// SIMATIC S7-200 project (STEP 7-Micro/WIN), CPU 226 REL 02.01

SYMBOL_TABLE 用户定义1
mAuto            I0.0     // 自动循环模式
mPosDirection    I0.1     // 正转方向
mRun             I1.1     // 启动
mStop            I1.3     // 停止
mStoped          I1.5     // 停止状态
rRunStop         Q0.0     // 启停输出K1
rDirection       Q0.2     // 方向输出K2
rBreak           Q0.5     // 制动输出K4
cmdRun           M0.2     // 运行指令
cmdDirPos        M0.3     // 方向指令1为正转
cmdModAuto       M0.4     // 手自动模式1为自动
TMP              M0.1
PosDuringAuto    M0.5     // 自动运行时切换方向触发
TMP1             M0.6
TMP2             M0.7
mAin             AIW0     // 用于设定时间的模拟量输入
END_SYMBOL_TABLE

SYMBOL_TABLE S7-200 符号
Always_On        SM0.0    // 始终接通为 ON
First_Scan_On    SM0.1    // 仅第一个扫描周期中接通为 ON
END_SYMBOL_TABLE

ORGANIZATION_BLOCK 主程序:OB1
TITLE=
VAR
AllTime:INT;	// LW0 
PosTime:INT;	// LW2 
END_VAR
BEGIN
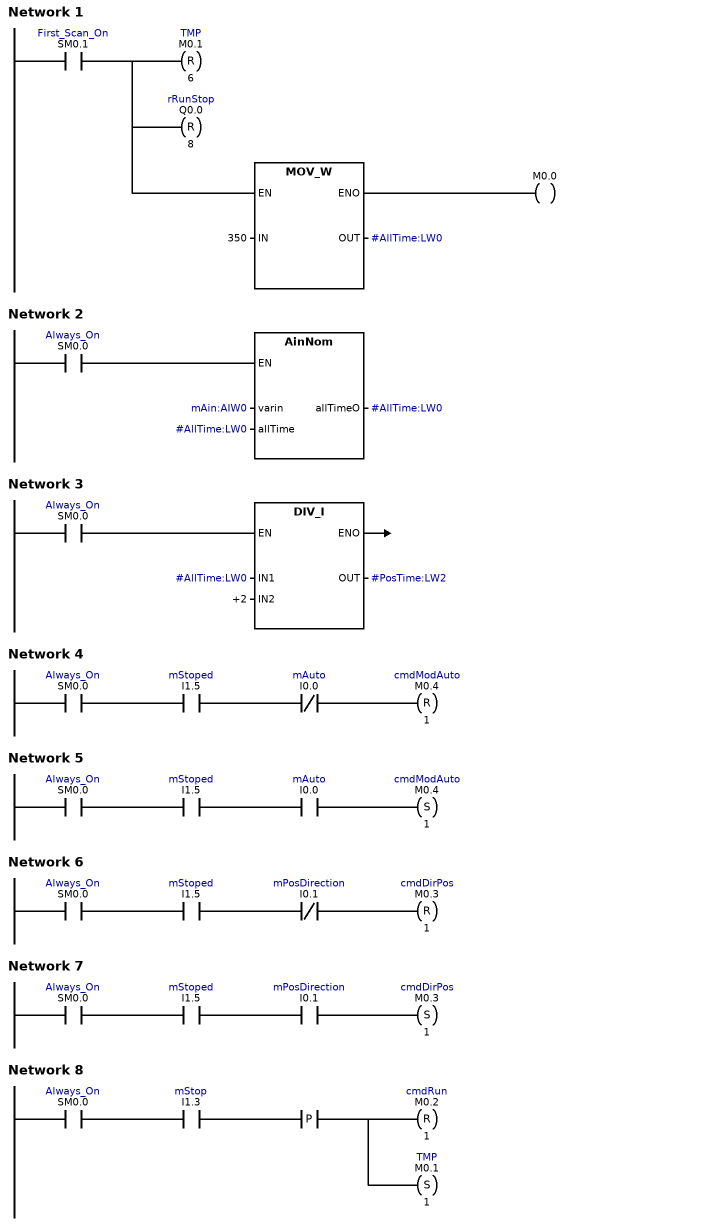
Network 1
LD     First_Scan_On:SM0.1
R      TMP:M0.1, 6
R      rRunStop:Q0.0, 8
MOVW   350, #AllTime:LW0
AENO
=      M0.0
Network 2
LD     Always_On:SM0.0
CALL   AinNom:SBR1, mAin:AIW0, #AllTime:LW0, #AllTime:LW0
Network 3
LD     Always_On:SM0.0
MOVW   #AllTime:LW0, #PosTime:LW2
/I     +2, #PosTime:LW2
Network 4
LD     Always_On:SM0.0
A      mStoped:I1.5
AN     mAuto:I0.0
R      cmdModAuto:M0.4, 1
Network 5
LD     Always_On:SM0.0
A      mStoped:I1.5
A      mAuto:I0.0
S      cmdModAuto:M0.4, 1
Network 6
LD     Always_On:SM0.0
A      mStoped:I1.5
AN     mPosDirection:I0.1
R      cmdDirPos:M0.3, 1
Network 7
LD     Always_On:SM0.0
A      mStoped:I1.5
A      mPosDirection:I0.1
S      cmdDirPos:M0.3, 1
Network 8
LD     Always_On:SM0.0
A      mStop:I1.3
EU
R      cmdRun:M0.2, 1
S      TMP:M0.1, 1
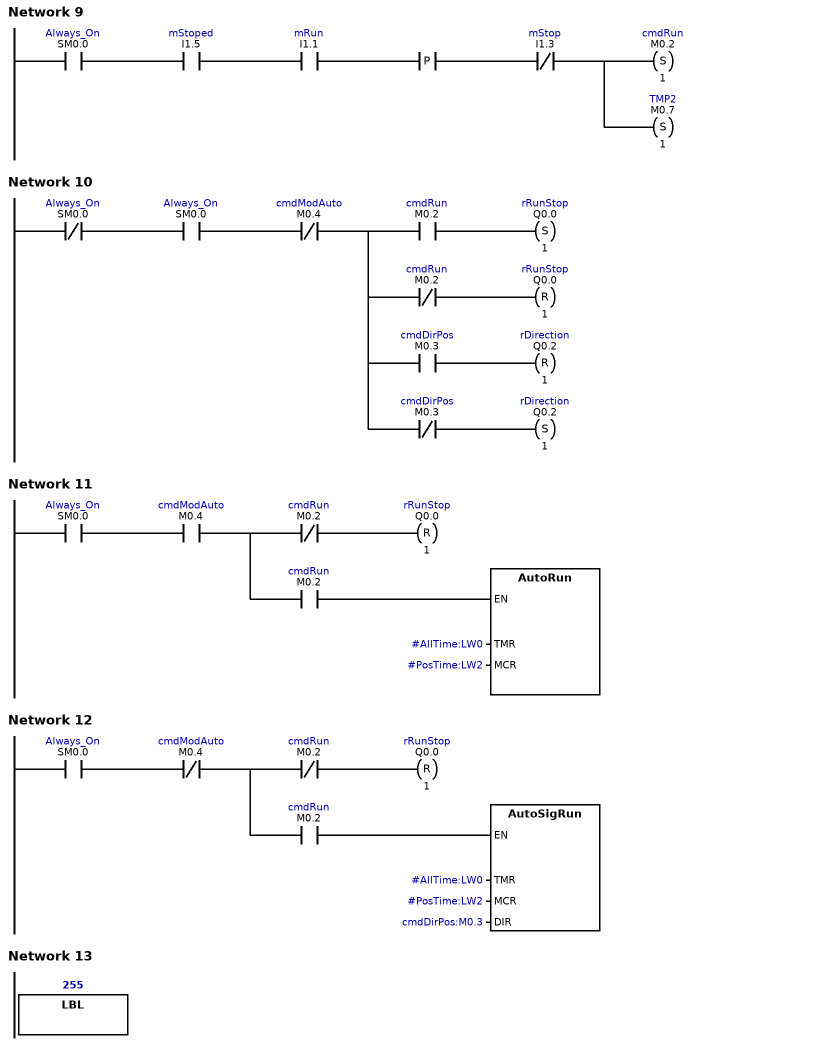
Network 9
LD     Always_On:SM0.0
A      mStoped:I1.5
A      mRun:I1.1
EU
AN     mStop:I1.3
S      cmdRun:M0.2, 1
S      TMP2:M0.7, 1
Network 10
LDN    Always_On:SM0.0
A      Always_On:SM0.0
AN     cmdModAuto:M0.4
LPS
A      cmdRun:M0.2
S      rRunStop:Q0.0, 1
LRD
AN     cmdRun:M0.2
R      rRunStop:Q0.0, 1
LRD
A      cmdDirPos:M0.3
R      rDirection:Q0.2, 1
LPP
AN     cmdDirPos:M0.3
S      rDirection:Q0.2, 1
Network 11
LD     Always_On:SM0.0
A      cmdModAuto:M0.4
LPS
AN     cmdRun:M0.2
R      rRunStop:Q0.0, 1
LPP
A      cmdRun:M0.2
CALL   AutoRun:SBR0, #AllTime:LW0, #PosTime:LW2
Network 12
LD     Always_On:SM0.0
AN     cmdModAuto:M0.4
LPS
AN     cmdRun:M0.2
R      rRunStop:Q0.0, 1
LPP
A      cmdRun:M0.2
CALL   AutoSigRun:SBR2, #AllTime:LW0, #PosTime:LW2, cmdDirPos:M0.3
Network 13
LBL    255
END_ORGANIZATION_BLOCK

SUBROUTINE_BLOCK AutoRun:SBR0
TITLE=子程序注释
VAR_INPUT
TMR:INT;	// LW0 
MCR:INT;	// LW2 
END_VAR
VAR
DET:INT;	// LW4 
END_VAR
BEGIN
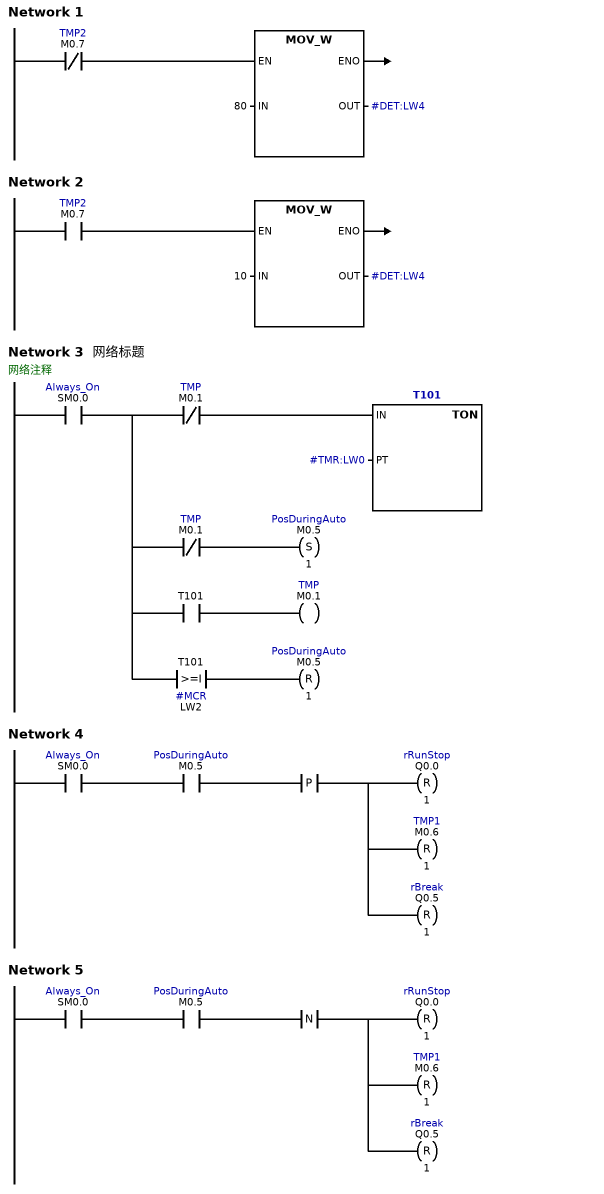
Network 1
LDN    TMP2:M0.7
MOVW   80, #DET:LW4
Network 2
LD     TMP2:M0.7
MOVW   10, #DET:LW4
Network 3 // 网络标题
// 网络注释
LD     Always_On:SM0.0
LPS
AN     TMP:M0.1
TON    T101, #TMR:LW0
LRD
AN     TMP:M0.1
S      PosDuringAuto:M0.5, 1
LRD
A      T101
=      TMP:M0.1
LPP
AW>=   T101, #MCR:LW2
R      PosDuringAuto:M0.5, 1
Network 4
LD     Always_On:SM0.0
A      PosDuringAuto:M0.5
EU
R      rRunStop:Q0.0, 1
R      TMP1:M0.6, 1
R      rBreak:Q0.5, 1
Network 5
LD     Always_On:SM0.0
A      PosDuringAuto:M0.5
ED
R      rRunStop:Q0.0, 1
R      TMP1:M0.6, 1
R      rBreak:Q0.5, 1
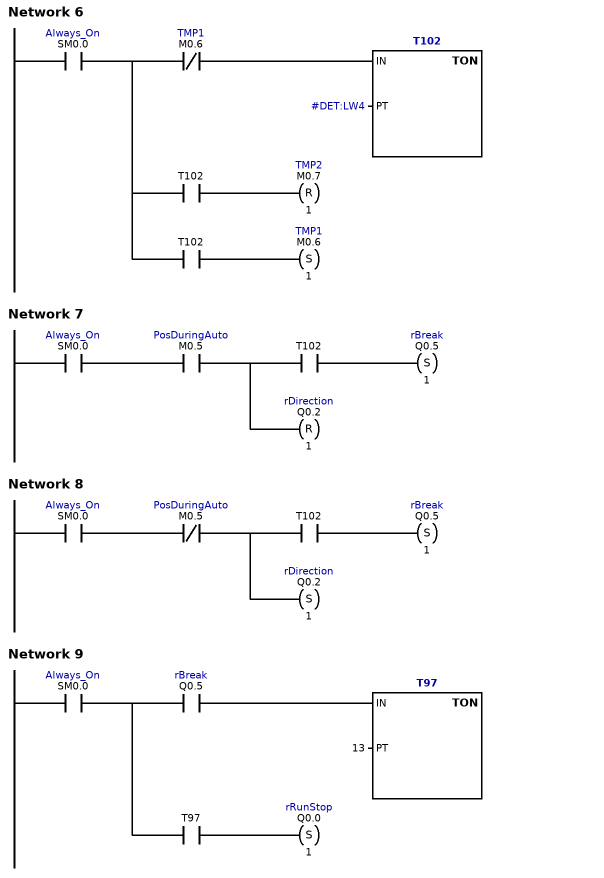
Network 6
LD     Always_On:SM0.0
LPS
AN     TMP1:M0.6
TON    T102, #DET:LW4
LRD
A      T102
R      TMP2:M0.7, 1
LPP
A      T102
S      TMP1:M0.6, 1
Network 7
LD     Always_On:SM0.0
A      PosDuringAuto:M0.5
LPS
A      T102
S      rBreak:Q0.5, 1
LPP
R      rDirection:Q0.2, 1
Network 8
LD     Always_On:SM0.0
AN     PosDuringAuto:M0.5
LPS
A      T102
S      rBreak:Q0.5, 1
LPP
S      rDirection:Q0.2, 1
Network 9
LD     Always_On:SM0.0
LPS
A      rBreak:Q0.5
TON    T97, 13
LPP
A      T97
S      rRunStop:Q0.0, 1
END_SUBROUTINE_BLOCK

SUBROUTINE_BLOCK AinNom:SBR1
TITLE=子程序注释
VAR_INPUT
varin:INT;	// LW0 
allTime:INT;	// LW2 
END_VAR
VAR_OUTPUT
allTimeO:INT;	// LW4 
END_VAR
BEGIN
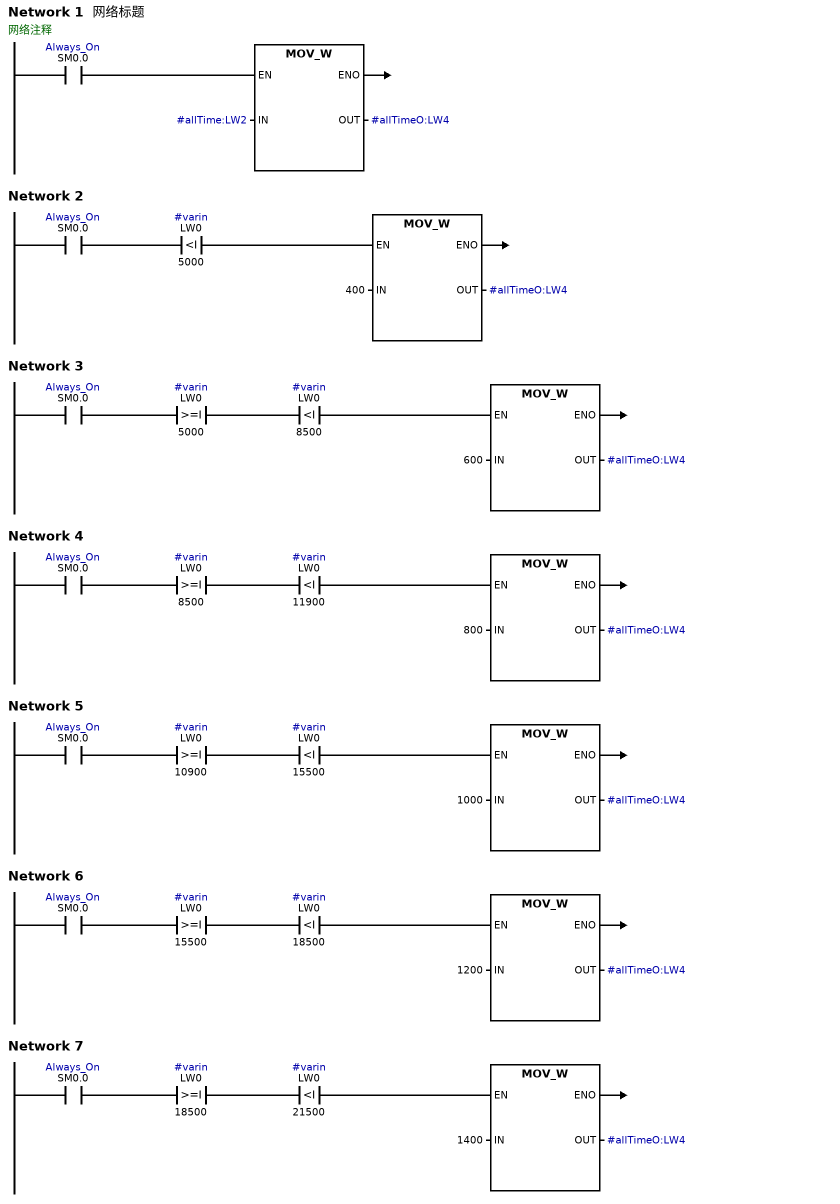
Network 1 // 网络标题
// 网络注释
LD     Always_On:SM0.0
MOVW   #allTime:LW2, #allTimeO:LW4
Network 2
LD     Always_On:SM0.0
AW<    #varin:LW0, 5000
MOVW   400, #allTimeO:LW4
Network 3
LD     Always_On:SM0.0
AW>=   #varin:LW0, 5000
AW<    #varin:LW0, 8500
MOVW   600, #allTimeO:LW4
Network 4
LD     Always_On:SM0.0
AW>=   #varin:LW0, 8500
AW<    #varin:LW0, 11900
MOVW   800, #allTimeO:LW4
Network 5
LD     Always_On:SM0.0
AW>=   #varin:LW0, 10900
AW<    #varin:LW0, 15500
MOVW   1000, #allTimeO:LW4
Network 6
LD     Always_On:SM0.0
AW>=   #varin:LW0, 15500
AW<    #varin:LW0, 18500
MOVW   1200, #allTimeO:LW4
Network 7
LD     Always_On:SM0.0
AW>=   #varin:LW0, 18500
AW<    #varin:LW0, 21500
MOVW   1400, #allTimeO:LW4
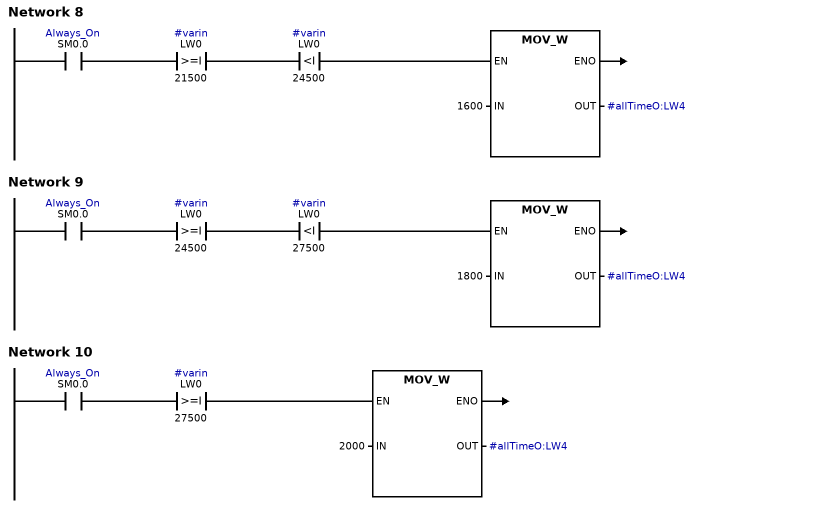
Network 8
LD     Always_On:SM0.0
AW>=   #varin:LW0, 21500
AW<    #varin:LW0, 24500
MOVW   1600, #allTimeO:LW4
Network 9
LD     Always_On:SM0.0
AW>=   #varin:LW0, 24500
AW<    #varin:LW0, 27500
MOVW   1800, #allTimeO:LW4
Network 10
LD     Always_On:SM0.0
AW>=   #varin:LW0, 27500
MOVW   2000, #allTimeO:LW4
END_SUBROUTINE_BLOCK

SUBROUTINE_BLOCK AutoSigRun:SBR2
TITLE=
VAR_INPUT
TMR:INT;	// LW0 
MCR:INT;	// LW2 
DIR:BOOL;	// L4.0 
END_VAR
VAR
DET:INT;	// LW5 
END_VAR
BEGIN
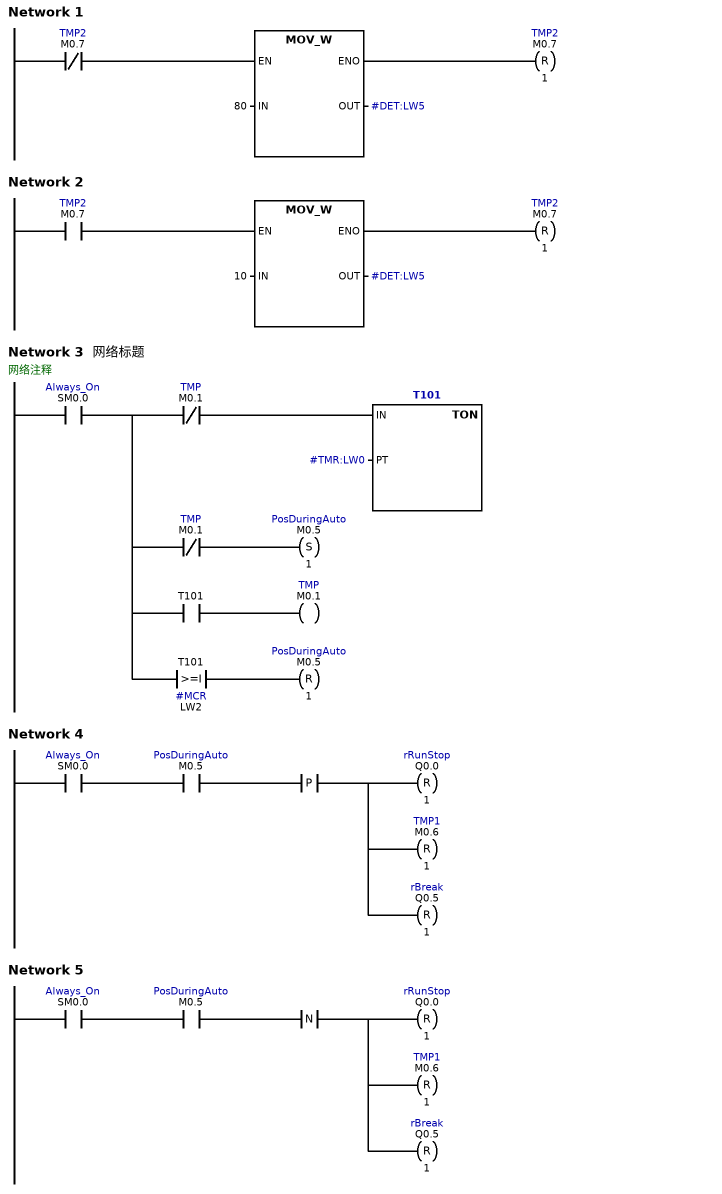
Network 1
LDN    TMP2:M0.7
MOVW   80, #DET:LW5
AENO
R      TMP2:M0.7, 1
Network 2
LD     TMP2:M0.7
MOVW   10, #DET:LW5
AENO
R      TMP2:M0.7, 1
Network 3 // 网络标题
// 网络注释
LD     Always_On:SM0.0
LPS
AN     TMP:M0.1
TON    T101, #TMR:LW0
LRD
AN     TMP:M0.1
S      PosDuringAuto:M0.5, 1
LRD
A      T101
=      TMP:M0.1
LPP
AW>=   T101, #MCR:LW2
R      PosDuringAuto:M0.5, 1
Network 4
LD     Always_On:SM0.0
A      PosDuringAuto:M0.5
EU
R      rRunStop:Q0.0, 1
R      TMP1:M0.6, 1
R      rBreak:Q0.5, 1
Network 5
LD     Always_On:SM0.0
A      PosDuringAuto:M0.5
ED
R      rRunStop:Q0.0, 1
R      TMP1:M0.6, 1
R      rBreak:Q0.5, 1
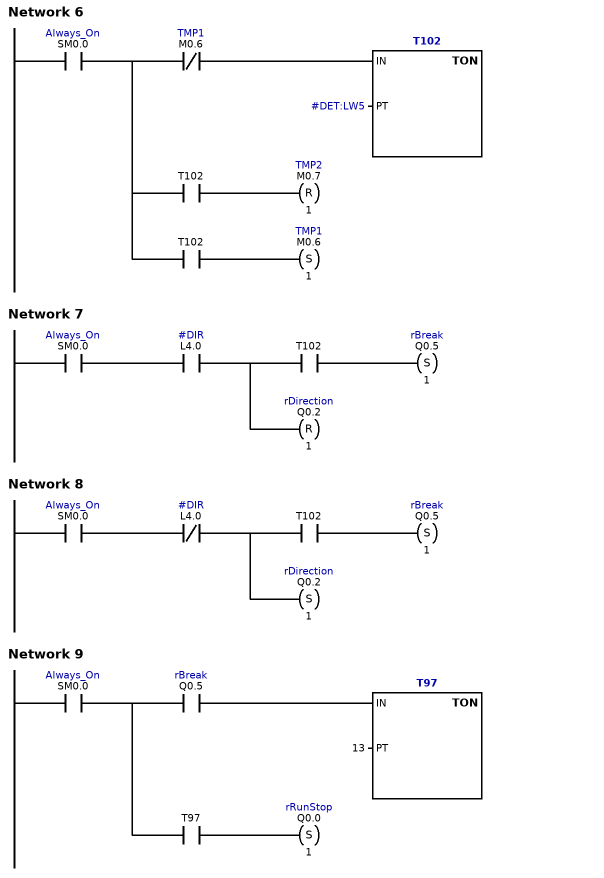
Network 6
LD     Always_On:SM0.0
LPS
AN     TMP1:M0.6
TON    T102, #DET:LW5
LRD
A      T102
R      TMP2:M0.7, 1
LPP
A      T102
S      TMP1:M0.6, 1
Network 7
LD     Always_On:SM0.0
A      #DIR:L4.0
LPS
A      T102
S      rBreak:Q0.5, 1
LPP
R      rDirection:Q0.2, 1
Network 8
LD     Always_On:SM0.0
AN     #DIR:L4.0
LPS
A      T102
S      rBreak:Q0.5, 1
LPP
S      rDirection:Q0.2, 1
Network 9
LD     Always_On:SM0.0
LPS
A      rBreak:Q0.5
TON    T97, 13
LPP
A      T97
S      rRunStop:Q0.0, 1
END_SUBROUTINE_BLOCK

DATA_BLOCK_TAB 用户定义1
BEGIN
//数据页注释
//按 F1 键获取帮助和示范数据页
VB0      255
VB1      255
VB2      255
END_DATA_BLOCK_TAB
